FUNCTION_BLOCK UNIT_OwnerView (* Subscribes to the unit's occupation owner (local channel) and asks for the current owner at INIT *)
  (* Standard: 61499-2 *)
  (* Version 0.1, 2026-09-28, Project contributors, AAU Smart Production Lab *)
  PACKAGE unitlib;
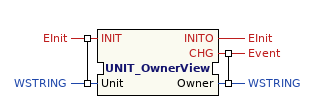
  EVENT_INPUT
    INIT : EInit WITH Unit;
  END_EVENT
  EVENT_OUTPUT
    INITO : EInit;
    CHG WITH Owner;
  END_EVENT
  VAR_INPUT
    Unit : WSTRING;
  END_VAR
  VAR_OUTPUT
    Owner : WSTRING;
  END_VAR
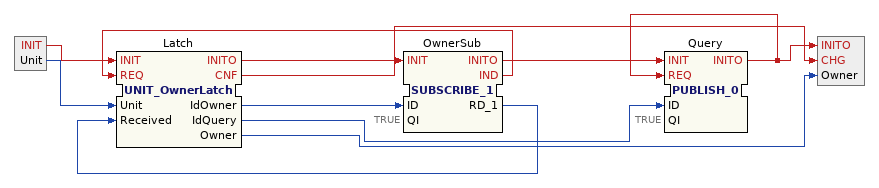
  FBS
    Latch : unitlib::UNIT_OwnerLatch;
    OwnerSub : iec61499::net::SUBSCRIBE_1(QI := TRUE);
    Query : iec61499::net::PUBLISH_0(QI := TRUE);
  END_FBS
  EVENT_CONNECTIONS
    INIT TO Latch.INIT;
    Latch.INITO TO OwnerSub.INIT;
    OwnerSub.INITO TO Query.INIT;
    Query.INITO TO Query.REQ;
    Query.INITO TO INITO;
    OwnerSub.IND TO Latch.REQ;
    Latch.CNF TO CHG;
  END_CONNECTIONS
  DATA_CONNECTIONS
    Unit TO Latch.Unit;
    Latch.IdOwner TO OwnerSub.ID;
    Latch.IdQuery TO Query.ID;
    OwnerSub.RD_1 TO Latch.Received;
    Latch.Owner TO Owner;
  END_CONNECTIONS
END_FUNCTION_BLOCK
